Fanuc TP program (LS listing): PNS0001.LS

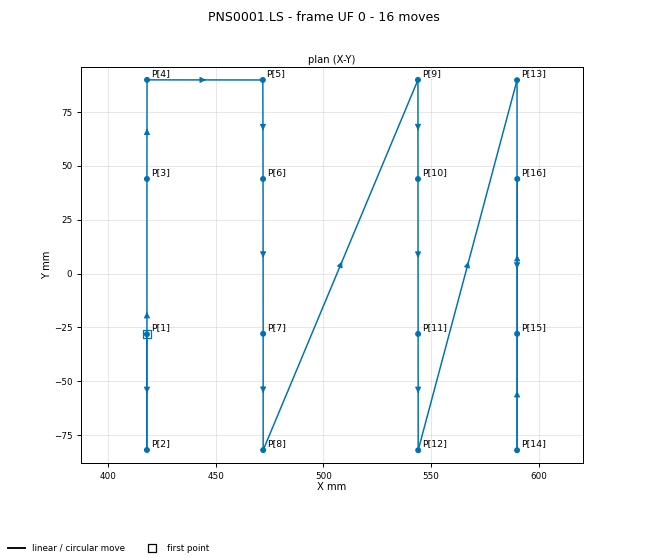
[picture p0: tool path of PNS0001.LS in frame UF 0, 16 of 16 moves have a stored position in this frame; points joined in program order, loops and branches not executed]
/PROG  PNS888
/ATTR
OWNER       = MNEDITOR;
COMMENT     = "";
PROG_SIZE   = 636;
CREATE      = DATE 23-01-07  TIME 11:59:14;
MODIFIED    = DATE 23-01-07  TIME 12:02:18;
FILE_NAME   = ;
VERSION     = 0;
LINE_COUNT  = 4;
MEMORY_SIZE = 992;
PROTECT     = READ_WRITE;
TCD:  STACK_SIZE	= 0,
      TASK_PRIORITY	= 50,
      TIME_SLICE	= 0,
      BUSY_LAMP_OFF	= 0,
      ABORT_REQUEST	= 0,
      PAUSE_REQUEST	= 0;
DEFAULT_GROUP	= 1,*,*,*,*;
CONTROL_CODE	= 00000000 00000000;
/MN
   1:J P[1] 100% FINE    ;
   2:L P[2] 100mm/sec CNT0    ;
   3:L P[3] 100mm/sec CNT0    ;
   4:L P[4] 100mm/sec CNT0    ;
   5:L P[5] 100mm/sec CNT0    ;
   6:L P[6] 100mm/sec CNT0    ;
   7:L P[7] 100mm/sec CNT0    ;
   8:L P[8] 100mm/sec CNT0    ;
   9:L P[9] 100mm/sec CNT0    ;
   10:L P[10] 100mm/sec CNT0    ;
   11:L P[11] 100mm/sec CNT0    ;
   12:L P[12] 100mm/sec CNT0    ;
   13:L P[13] 100mm/sec CNT0    ;
   14:L P[14] 100mm/sec CNT0    ;
   15:L P[15] 100mm/sec CNT0    ;
   16:L P[16] 100mm/sec CNT0    ;
/POS
P[1]{
   GP1:
	UF : 0, UT : 1,		CONFIG : 'N U T, 0, 0, 0',
	X =  417.991  mm,	Y =   -28.157  mm,	Z =   -270.000  mm,
	W =  0.000 deg,	P =   0.000 deg,	R =   1.000 deg
};
P[2]{
   GP1:
	UF : 0, UT : 1,		CONFIG : 'N U T, 0, 0, 0',
	X =  417.993  mm,	Y =   -81.917  mm,	Z =   -270.000  mm,
	W =  0.000 deg,	P =   0.000 deg,	R =   1.000 deg
};
P[3]{
   GP1:
	UF : 0, UT : 1,		CONFIG : 'N U T, 0, 0, 0',
	X =  418.000  mm,	Y =   43.985  mm,	Z =   -270.000  mm,
	W =  0.000 deg,	P =   0.000 deg,	R =   1.000 deg
};
P[4]{
   GP1:
	UF : 0, UT : 1,		CONFIG : 'N U T, 0, 0, 0',
	X =  418.044  mm,	Y =   90.015  mm,	Z =   -270.000  mm,
	W =  0.000 deg,	P =   0.000 deg,	R =   1.000 deg
};
P[5]{
   GP1:
	UF : 0, UT : 1,		CONFIG : 'N U T, 0, 0, 0',
	X =  471.835  mm,	Y =   89.959  mm,	Z =   -270.000  mm,
	W =  0.000 deg,	P =   0.000 deg,	R =   1.000 deg
};
P[6]{
   GP1:
	UF : 0, UT : 1,		CONFIG : 'N U T, 0, 0, 0',
	X =  471.940  mm,	Y =   43.979  mm,	Z =   -270.000  mm,
	W =  0.000 deg,	P =   0.000 deg,	R =   1.000 deg
};
P[7]{
   GP1:
	UF : 0, UT : 1,		CONFIG : 'N U T, 0, 0, 0',
	X =  471.980  mm,	Y =   -27.930  mm,	Z =   -270.000  mm,
	W =  0.000 deg,	P =   0.000 deg,	R =   1.000 deg
};
P[8]{
   GP1:
	UF : 0, UT : 1,		CONFIG : 'N U T, 0, 0, 0',
	X =  471.992  mm,	Y =   -81.959  mm,	Z =   -270.000  mm,
	W =  0.000 deg,	P =   0.000 deg,	R =   1.000 deg
};
P[9]{
   GP1:
	UF : 0, UT : 1,		CONFIG : 'N U T, 0, 0, 0',
	X =  543.896  mm,	Y =   90.001  mm,	Z =   -270.000  mm,
	W =  -0.000 deg,	P =   -0.000 deg,	R =   1.000 deg
};
P[10]{
   GP1:
	UF : 0, UT : 1,		CONFIG : 'N U T, 0, 0, 0',
	X =  543.904  mm,	Y =   43.962  mm,	Z =   -270.000  mm,
	W =  -0.000 deg,	P =   0.000 deg,	R =   1.000 deg
};
P[11]{
   GP1:
	UF : 0, UT : 1,		CONFIG : 'N U T, 0, 0, 0',
	X =  543.962  mm,	Y =   -28.007  mm,	Z =   -270.000  mm,
	W =  0.000 deg,	P =   0.000 deg,	R =   1.000 deg
};
P[12]{
   GP1:
	UF : 0, UT : 1,		CONFIG : 'N U T, 0, 0, 0',
	X =  543.997  mm,	Y =   -82.039  mm,	Z =   -270.000  mm,
	W =  0.000 deg,	P =   0.000 deg,	R =   1.000 deg
};
P[13]{
   GP1:
	UF : 0, UT : 1,		CONFIG : 'N U T, 0, 0, 0',
	X =  589.921  mm,	Y =   89.879  mm,	Z =   -270.000  mm,
	W =  -0.000 deg,	P =   0.000 deg,	R =   1.000 deg
};
P[14]{
   GP1:
	UF : 0, UT : 1,		CONFIG : 'N U T, 0, 0, 0',
	X =  589.927  mm,	Y =   -82.042  mm,	Z =   -270.000  mm,
	W =  0.000 deg,	P =   0.000 deg,	R =   1.000 deg
};
P[15]{
   GP1:
	UF : 0, UT : 1,		CONFIG : 'N U T, 0, 0, 0',
	X =  589.955  mm,	Y =   -27.942  mm,	Z =   -270.000  mm,
	W =  0.000 deg,	P =   0.000 deg,	R =   1.000 deg
};
P[16]{
   GP1:
	UF : 0, UT : 1,		CONFIG : 'N U T, 0, 0, 0',
	X =  590.031  mm,	Y =   43.979  mm,	Z =   -270.000  mm,
	W =  -0.000 deg,	P =   -0.000 deg,	R =   1.000 deg
};
/END
